FUNCTION_BLOCK TExecution_EventHandler // Event Handler used to check that TExecution raises events correctly
IMPLEMENTS
    IEventHandler_OnExecutionAborted,
    IEventHandler_OnExecutionFailed
VAR_INPUT
END_VAR
VAR_OUTPUT
END_VAR
VAR
    _AbortedEventRaised : BOOL;
    _FailedEventRaised : BOOL;
    _EventMessage : T_MaxString;
END_VAR

PROPERTY AbortedEventRaised : BOOL
GET
AbortedEventRaised := _AbortedEventRaised;
END_GET
SET
_AbortedEventRaised := AbortedEventRaised;
END_SET
END_PROPERTY

PROPERTY FailedEventRaised : BOOL
GET
FailedEventRaised := _FailedEventRaised;
END_GET
SET
_FailedEventRaised := FailedEventRaised;
END_SET
END_PROPERTY

METHOD OnExecutionAborted
VAR_INPUT
	Message : T_MaxString;
END_VAR
_AbortedEventRaised := TRUE;
_EventMessage := Message;
END_METHOD

METHOD OnExecutionFailed
VAR_INPUT
	Message : T_MaxString;
END_VAR
_FailedEventRaised := TRUE;
_EventMessage := Message;
END_METHOD

END_FUNCTION_BLOCK

(* stored: Version 1.1.0.1, ProductVersion 3.1.4024.4
   POU TExecution_EventHandler: Id {f6b89d26-f417-4707-9332-e9ff274e933f}, SpecialFunc None
   Property AbortedEventRaised: Id {141dc362-1fda-4648-a009-66ff4621876d}
   Get Get: Id {b1751aa5-823a-40f1-a481-b5fda573e0a0}
   Set Set: Id {2a8b9752-82fe-4f88-b969-9a7388e1b328}
   Property FailedEventRaised: Id {789ca6bd-d8db-4976-8414-9cdbc9cc0f62}
   Get Get: Id {23c589a3-4d6b-4963-a5e1-aa0cf220f357}
   Set Set: Id {fb1649e4-0442-45ce-a028-602e4b9edb41}
   Method OnExecutionAborted: Id {09c9a637-0904-45d1-b185-d66b533fe6f4}
   Method OnExecutionFailed: Id {6e8ba4db-2d8f-4121-a6d3-1366cdb13c6a} *)
